TYPE ST_APP_STATE :
STRUCT
  AppState            : E_INSTANCE_STATE;
  InstanceStates      : REFERENCE TO ARRAY[1..MAX_PROCESS] OF ST_INSTANCE_STATE;
  XtsTransportState   : REFERENCE TO ST_XTS_TRANSPORT_STATE;
END_STRUCT
END_TYPE

(* stored: Version 1.1.0.1, ProductVersion 3.1.4024.15
   DUT ST_APP_STATE: Id {8ad5dcc9-9492-4d8e-972f-a2d6ca9938d0} *)
